AssertTrue(q_Output,
    'Beam within limits, FFO should be true');
    
    
//Req eV moved out of range
stCurBeamParams.neVRange := F_eVRangeCalculator(800, 0);
    
stMachineTargetBeamParams.neVRange := F_eVRangeCalculator(800, 0);

stReqBeamParams.neVRange := 2#0000_1111_0011_1111;

fbPEW.i_xReset := FALSE; //release local FF reset req    
fbPEW(i_stCurrentBeamParams := stCurBeamParams,
    i_stMachineTargetBeamParams := stMachineTargetBeamParams,
    i_stRequestedBeamParams := stReqBeamParams,
    io_fbFFHWO := fbFFO);
    
fbFFO.EvaluateOutput(q_xFastFaultOut=>q_Output);

AssertFalse(q_Output,
    'Limits moved beyond current and target beam, should produce a fault.');

//Beam and target eV moved back within permitted ranges, reset clears fault
stCurBeamParams.neVRange := F_eVRangeCalculator( 300, 0);
    
stMachineTargetBeamParams.neVRange := F_eVRangeCalculator(300, 0);

stReqBeamParams.neVRange := 2#0000_1111_0011_1111;

fbFFO(i_xReset:=TRUE); //New reset request

fbPEW.i_xReset := TRUE; //New reset request

fbPEW(i_stCurrentBeamParams := stCurBeamParams, //Beam params are now within spec
    i_stMachineTargetBeamParams := stMachineTargetBeamParams,
    i_stRequestedBeamParams := stReqBeamParams,
    io_fbFFHWO := fbFFO);
    
fbFFO.EvaluateOutput(q_xFastFaultOut=>q_Output);

AssertTrue(q_Output,
    'Beam within limits after reset, FFO should be true');
    
//At this point, the fast fault would be cleared

//Current beam eV moved out of range
stCurBeamParams.neVRange := F_eVRangeCalculator(800, 0); //Moved out of range
    
stMachineTargetBeamParams.neVRange := F_eVRangeCalculator(300, 0); //Still within range

stReqBeamParams.neVRange := 2#0000_1111_0011_1111;

fbPEW(i_stCurrentBeamParams := stCurBeamParams,
    i_stMachineTargetBeamParams := stMachineTargetBeamParams,
    i_stRequestedBeamParams := stReqBeamParams,
    io_fbFFHWO := fbFFO);
    
fbFFO.EvaluateOutput(q_xFastFaultOut=>q_Output);

AssertFalse(q_Output,
    'Current beam moved beyond set limits, should produce a fault');

//Target beam eV moved out of range
fbFFO(i_xReset:=FALSE); //Reset released
fbFFO(i_xReset:=TRUE); //New reset request comes in at the top of a cycle, but will be overridden

stCurBeamParams.neVRange := F_eVRangeCalculator(300, 0); //Now within range
    
stMachineTargetBeamParams.neVRange := F_eVRangeCalculator(800, 0); //Moved out of range

stReqBeamParams.neVRange := 2#0000_1111_0011_1111;

fbPEW.i_xReset := TRUE; //Attempt to reset local FF will fail
fbPEW(i_stCurrentBeamParams := stCurBeamParams,
    i_stMachineTargetBeamParams := stMachineTargetBeamParams,
    i_stRequestedBeamParams := stReqBeamParams,
    io_fbFFHWO := fbFFO);
    
fbFFO.EvaluateOutput(q_xFastFaultOut=>q_Output);

AssertFalse(q_Output,
    'Target beam moved beyond set limits, should produce a fault');
    
TEST_FINISHED();
END_METHOD

END_FUNCTION_BLOCK

// TestComponents/FB_SafeBPCompare_Test
{attribute 'call_after_init'}
FUNCTION_BLOCK FB_SafeBPCompare_Test EXTENDS TcUnit.FB_TestSuite
VAR_INPUT
END_VAR
VAR_OUTPUT
END_VAR
VAR

END_VAR

BeamOffIsSafe();
BPComparisonCheck();

//Verify beam off is considered safe.
METHOD BeamOffIsSafe
VAR_INPUT
END_VAR
VAR
    stBeamOn_MoreConservative    :    ST_BeamParams;
    stBeamOff_LessConservative    :    ST_BeamParams;
END_VAR
stBeamOn_MoreConservative  := F_SetBeamParams(
    0, //0% transmission is more conservative than 50
    16#FFFF_FFFF,
    120, //rate
    PMPS_GVL.DUMMY_AUX_ATT_ARRAY);

stBeamOff_LessConservative:= F_SetBeamParams(
    0.5, //50% transmission, less conservative, without 0-rate this beam parameter set would be less safe than above
    16#FFFF_FFFF,
    0, //rate, hence, more conservative
    PMPS_GVL.DUMMY_AUX_ATT_ARRAY); //0 beam rate means this bps is actually safer than BeamOn

TEST('BeamOffIsSafe');
    
AssertTrue(
    F_SafeBPCompare0Rate(stBeamOff_LessConservative, stBeamOn_MoreConservative),
    'SafeBPCompare does not think beam rate = 0 is safer than anything else.'); 
TEST_FINISHED();
END_METHOD

//Verify BP comparison remains logical.
METHOD BPComparisonCheck
VAR_INPUT
END_VAR
VAR
    stSafer    :    ST_BeamParams;
    stNotSoSafe    :    ST_BeamParams;
    idx : UINT;
    
    xResult : BOOL;
    xFailedTest : BOOL; // To exit loops early
END_VAR

TEST('BPComparisonTran');
//Attenuation
stSafer := F_SetBeamParams(
    0.51, //
    16#FFFFFFFF,
    1,
    PMPS_GVL.DUMMY_AUX_ATT_ARRAY);

stNotSoSafe := F_SetBeamParams(
    0.61, //
    16#FFFFFFFF,
    1,
    PMPS_GVL.DUMMY_AUX_ATT_ARRAY); 
    
AssertTrue(
    F_SafeBPCompare(stSafer, stNotSoSafe),
    'Attenuation eval is broken (True)'); 

AssertFalse(
    F_SafeBPCompare(stNotSoSafe, stSafer),
    'Attenuation eval is broken (False)');
    
// Check at margin threshold
stSafer.nTran := stNotSoSafe.nTran*(PMPS_GVL.TRANS_SCALING_FACTOR + PMPS_PARAM.TRANS_MARGIN)/PMPS_GVL.TRANS_SCALING_FACTOR;
AssertTrue(
    F_SafeBPCompare(stSafer, stNotSoSafe),
    'Attenuation eval is broken: should be safe up to margin.');

stSafer.nTran := 1 + stNotSoSafe.nTran*(PMPS_GVL.TRANS_SCALING_FACTOR + PMPS_PARAM.TRANS_MARGIN)/PMPS_GVL.TRANS_SCALING_FACTOR;

AssertFalse(
    F_SafeBPCompare(stSafer, stNotSoSafe),
    'Attenuation eval is broken (False): should not be safe at all past margin');

TEST_FINISHED();


    
//Attenuator array    
TEST('BPComparisonTranArray');

stSafer := F_SetBeamParams(
    0, //
    16#FFFFFFFF,
    1,
    PMPS_GVL.DUMMY_AUX_ATT_ARRAY); 

stNotSoSafe := F_SetBeamParams(
    0, //
    16#FFFFFFFF,
    1,
    PMPS_GVL.DUMMY_AUX_ATT_ARRAY); 

FOR idx:=1 TO PMPS_GVL.AUX_ATTENUATORS DO
    stSafer.astAttenuators[idx].nTran := 0.00500;
    stNotSoSafe.astAttenuators[idx].nTran := 0.00600;
    
    xResult := F_SafeBPCompare(stSafer, stNotSoSafe);
    
    AssertTrue(
    xResult,
    'Attenuation array eval is broken (True)');
 
    xFailedTest S= NOT xResult;
    
    xResult := F_SafeBPCompare(stNotSoSafe, stSafer);
    AssertFalse(
    xResult,
    'Attenuation array eval is broken (False)');
    
    xFailedTest S= xResult;
    
    // Check at margin threshold
        stSafer.astAttenuators[idx].nTran := stNotSoSafe.astAttenuators[idx].nTran*(PMPS_GVL.TRANS_SCALING_FACTOR + PMPS_PARAM.TRANS_MARGIN)/PMPS_GVL.TRANS_SCALING_FACTOR;
        
        xResult := F_SafeBPCompare(stSafer, stNotSoSafe);
    
        AssertTrue(
            xResult,
            'Attenuation eval is broken: should be safe up to margin.');
        xFailedTest S= NOT xResult;
            
        stSafer.astAttenuators[idx].nTran := 1 + stNotSoSafe.astAttenuators[idx].nTran*(PMPS_GVL.TRANS_SCALING_FACTOR + PMPS_PARAM.TRANS_MARGIN)/PMPS_GVL.TRANS_SCALING_FACTOR;
        
        xResult := F_SafeBPCompare(stSafer, stNotSoSafe);
        AssertFalse(
            xResult,
            'Attenuation eval is broken (False): should not be safe at all past margin');
        xFailedTest S= xResult;
    //////////////////////
    IF xFailedTest THEN
        stSafer.astAttenuators[idx].nTran := 0;
        stNotSoSafe.astAttenuators[idx].nTran := 0;
        xFailedTest := FALSE;
        EXIT; // Exit this loop on the first failure.
	END_IF
    
    stSafer.astAttenuators[idx].nTran := 0;
    stNotSoSafe.astAttenuators[idx].nTran := 0;
    
END_FOR

TEST_FINISHED();

stSafer.astAttenuators[idx].nTran := 0;
stNotSoSafe.astAttenuators[idx].nTran := 0;

//Aperture array
TEST('BPComparisonApertureArray');

FOR idx:=1 TO PMPS_GVL.MAX_APERTURES DO
    // Height
    stSafer.astApertures[idx].Height := 30; // narrower is safer
    stNotSoSafe.astApertures[idx].Height := 50;
    
    AssertTrue(
    F_SafeBPCompare(stSafer, stNotSoSafe),
    'Aperture array eval is broken on height (True)'); 

    AssertFalse(
    F_SafeBPCompare(stNotSoSafe, stSafer),
    'Aperture array eval is broken on height (False)');
    
    IF NOT F_SafeBPCompare(stSafer, stNotSoSafe) or F_SafeBPCompare(stNotSoSafe, stSafer) THEN
        EXIT; // Exit this loop on the first failure.
	END_IF
    
    stSafer.astApertures[idx].Height := 0;
    stNotSoSafe.astApertures[idx].Height := 0;
    
    // Width
    stSafer.astApertures[idx].Width := 30; // narrower is safer
    stNotSoSafe.astApertures[idx].Width := 50;
    
    AssertTrue(
    F_SafeBPCompare(stSafer, stNotSoSafe),
    'Aperture array eval is broken on width (True)'); 

    AssertFalse(
    F_SafeBPCompare(stNotSoSafe, stSafer),
    'Aperture array eval is broken on width (False)');
    
    IF NOT F_SafeBPCompare(stSafer, stNotSoSafe) or F_SafeBPCompare(stNotSoSafe, stSafer) THEN
        EXIT; // Exit this loop on the first failure.
	END_IF
    
    stSafer.astApertures[idx].Width := 0;
    stNotSoSafe.astApertures[idx].Width := 0;
    
    
END_FOR

TEST_FINISHED();
    
//Rate
TEST('BPComparisonRate');
stSafer := F_SetBeamParams(
    0,
    16#FFFF_FFFF,
    1,
    PMPS_GVL.DUMMY_AUX_ATT_ARRAY); //

stNotSoSafe := F_SetBeamParams(
    0,
    16#FFFF_FFFF,
    10,
    PMPS_GVL.DUMMY_AUX_ATT_ARRAY); //
    
AssertTrue(
    F_SafeBPCompare(stSafer, stNotSoSafe),
    'Rate eval is broken (True)'); 

AssertFalse(
    F_SafeBPCompare(stNotSoSafe, stSafer),
    'Rate eval is broken (False)');
TEST_FINISHED();
    
//Pulse energy
(*
TEST('BPComparisonPulseEnergy');
stSafer := F_SetBeamParams(
    0, 
    1, //
    16#FFFF,
    1,
    PMPS_GVL.DUMMY_AUX_ATT_ARRAY);

stNotSoSafe := F_SetBeamParams(
    0, 
    10, //
    16#FFFF,
    1,
    PMPS_GVL.DUMMY_AUX_ATT_ARRAY); 
    *)
AssertTrue(
    F_SafeBPCompare(stSafer, stNotSoSafe),
    'Pulse energy eval is broken (True)'); 

AssertFalse(
    F_SafeBPCompare(stNotSoSafe, stSafer),
    'Pulse energy eval is broken (False)');    
TEST_FINISHED();
    
//Photon energy
//More extensive tests elsewhere
TEST('BPComparisonPhotonEnergy');
stSafer := F_SetBeamParams(
    0, 
    2#0000_0000_0000_0000_0000_0000_0000_0010,
    1,
    PMPS_GVL.DUMMY_AUX_ATT_ARRAY);

stNotSoSafe := F_SetBeamParams(
    0, 
    2#0000_0000_0000_0000_0000_0000_0000_0110,
    1,
    PMPS_GVL.DUMMY_AUX_ATT_ARRAY);
    
AssertTrue(
    F_SafeBPCompare(stSafer, stNotSoSafe),
    'Photon energy eval is broken (True)'); 

AssertFalse(
    F_SafeBPCompare(stNotSoSafe, stSafer),
    'Photon energy eval is broken (False)');    
TEST_FINISHED();
END_METHOD

END_FUNCTION_BLOCK

// TestComponents/FB_SubsysToArb_Test
{attribute 'call_after_init'}
FUNCTION_BLOCK FB_SubsysToArb_Test EXTENDS TcUnit.FB_TestSuite
VAR_INPUT
END_VAR
VAR_OUTPUT
END_VAR
VAR
END_VAR

BasicFunction();
VetoFunction();

METHOD BasicFunction
VAR_INPUT
END_VAR
VAR   
    nId    :    DWORD := 1;
    stReq    :    ST_BeamParams := (nTran:=12);
END_VAR
VAR_INST
    fbArbiter    :    FB_Arbiter(1);
    
    fbSubSysToArb : FB_SubSysToArbiter_IO; // Subsystem interface with beamline arbiter PLC
    pBPC : POINTER TO ST_BeamParams_IO;
    
    ioCurrentBP : ST_BeamParams_IO; 
    
    FFO : FB_HardwareFFOutput; // Dummy FFO not important for these tests
    
    nCohortScratch : UDINT;
    
END_VAR
VAR CONSTANT
    SysID : DWORD := 42;
END_VAR
// This simulates a synchronous cycle between the subsystem and arbiter PLC cycles. Ie. phase is locked, and cycle time is the same. This is not always the case, so these tests should be 
// trusted with a grain of salt.

TEST('Add to arbiter');

IF NOT fbArbiter.CheckRequestInPool(nID) THEN
    AssertTrue(fbArbiter.AddRequest(nId, stReq,'Device'), 'Arbiter returned false from AddRequest'); // some device asking its local arbiter for some beam parameters
END_IF  
   
TEST_FINISHED();   

///////////////////////////////////////
//Sub system cycle
fbSubSysToArb(Arbiter := fbArbiter, fbFFHWO := FFO);
//END of sub system cycle
///////////////////////////////////////


TEST('Initial Elevation');
AssertTrue(fbSubSysToArb.nRequestCohort = fbSubSysToArb.q_stRequestedBP.nCohortInt, 'ReqCohort and qBP Cohort do not match');
AssertFalse(fbArbiter.nActiveCohort <> 0, 'Arbiter indicates it is included in arbitration prematurely');
AssertTrue(fbSubSysToArb.nRequestCohort <> 0, 'Cohort index should move to 1 with first request');
TEST_FINISHED_NAMED('Initial Elevation');

nCohortScratch := fbSubSysToArb.nRequestCohort;
    
//Ethercat transfer simulation
// Transfer of requested BP to arbiter PLC
// pBPR := ADR(fbArbToSubSys.i_RequestedBP);
// pBPR^ := fbSubSysToArb.q_stRequestedBP;

ioCurrentBP := fbSubSysToArb.q_stRequestedBP;
// NOTE: Setting the returning cohort number to something less than the request cohort number
// will prevent the sub system arbiter FB from considering itself active in arbitration.
// The next set of tests verify this.
ioCurrentBP.nCohortInt := 0;

// Transfer of current BP to sub system PLC
pBPC := ADR(fbSubSysToArb.i_stCurrentBP);
pBPC^ := ioCurrentBP;

///////////////////////////////////////
//Sub system cycle
fbSubSysToArb(Arbiter := fbArbiter, fbFFHWO := FFO);
//END of sub system cycle
///////////////////////////////////////

TEST('Not yet active in arbitration');
AssertTrue(fbSubSysToArb.nActiveCohort = 0, 'Active cohort should still be zero, per ioCurrentBP.nCohortInt setting above.');
AssertFalse(fbArbiter.nActiveCohort <> 0, 'Arbiter indicates it is included in arbitration prematurely, checkrequest might be broken');
AssertTrue(fbSubSysToArb.nRequestCohort = nCohortScratch, 'Cohort index should not have changed because there have been no additional requests added to the arbiter');
TEST_FINISHED_NAMED('Not yet active in arbitration');

//Ethercat transfer simulation
// Transfer of requested BP to arbiter PLC
// pBPR := ADR(fbArbToSubSys.i_RequestedBP);
// pBPR^ := fbSubSysToArb.q_stRequestedBP;

ioCurrentBP := fbSubSysToArb.q_stRequestedBP;
// NOTE: Now we simulate the FB_ArbiterToSubSys_IO updating the cohort number to the same value as the request cohort, indicating that cohort has been included
ioCurrentBP.nCohortInt := 2;

// Transfer of current BP to sub system PLC
pBPC := ADR(fbSubSysToArb.i_stCurrentBP);
pBPC^ := ioCurrentBP;

///////////////////////////////////////
//Sub system cycle
fbSubSysToArb(Arbiter := fbArbiter, fbFFHWO := FFO);
//END of sub system cycle
///////////////////////////////////////

TEST('Active in arbitration');
AssertTrue(fbSubSysToArb.nActiveCohort = fbSubSysToArb.nRequestCohort, 'Active cohort and request cohort do not match');
AssertTrue(fbArbiter.nActiveCohort = 1, 'Arbiter does not indicate it is included in higher arbitration');
TEST_FINISHED_NAMED('Active in arbitration');
END_METHOD

METHOD VetoFunction
VAR_INPUT
END_VAR
VAR   
    nId    :    DWORD := 1;
    stReq    :    ST_BeamParams := (nTran:=12);
END_VAR
VAR_INST
    fbArbiter    :    FB_Arbiter(1);
    
    fbSubSysToArb : FB_SubSysToArbiter_IO; // Subsystem interface with beamline arbiter PLC
    fbArbToSubSys : FB_ArbiterToSubSys_IO;
    
    pBPC : POINTER TO ST_BeamParams_IO;
    pBPR : POINTER TO ST_BeamParams_IO;
    
    ioCurrentBP : ST_BeamParams_IO; 
    
    FFO : FB_HardwareFFOutput; // Dummy FFO not important for these tests
    
END_VAR
VAR CONSTANT
    SysID : DWORD := 42;
END_VAR
// This simulates a synchronous cycle between the subsystem and arbiter PLC cycles. Ie. phase is locked, and cycle time is the same. This is not always the case, so these tests should be 
// trusted with a grain of salt.

fbArbiter.AddRequest(nId, stReq,'Device'); // some device asking its local arbiter for some beam parameters


///////////////////////////////////////
//Sub system cycle
fbSubSysToArb(Arbiter := fbArbiter, fbFFHWO := FFO);
//END of sub system cycle
///////////////////////////////////////

TEST('Request propagated');
    AssertTrue(fbSubSysToArb.q_stRequestedBP.nTran = stReq.nTran, 'Request not propagated');
TEST_FINISHED();

// Veto activated
///////////////////////////////////////
//Sub system cycle
fbSubSysToArb(Arbiter := fbArbiter, fbFFHWO := FFO, i_bVeto:=TRUE);
//END of sub system cycle
///////////////////////////////////////

// Veto activated
///////////////////////////////////////
//Sub system cycle
fbSubSysToArb(Arbiter := fbArbiter, fbFFHWO := FFO, i_bVeto:=TRUE);
//END of sub system cycle
///////////////////////////////////////

TEST('Request sustained');
    AssertTrue(fbSubSysToArb.q_stRequestedBP.nTran = PMPS_GVL.cstFullBeam.nTran, 'Request still being propagated');
    AssertTrue(fbArbiter.CheckRequest(nId), 'Request still not valid');
TEST_FINISHED();

// Veto activated
///////////////////////////////////////
//Sub system cycle
fbSubSysToArb(Arbiter := fbArbiter, fbFFHWO := FFO, i_bVeto:=FALSE);
//END of sub system cycle
///////////////////////////////////////

// Veto activated
///////////////////////////////////////
//Sub system cycle
fbSubSysToArb(Arbiter := fbArbiter, fbFFHWO := FFO, i_bVeto:=FALSE);
fbSubSysToArb(Arbiter := fbArbiter, fbFFHWO := FFO, i_bVeto:=FALSE);
fbSubSysToArb(Arbiter := fbArbiter, fbFFHWO := FFO, i_bVeto:=FALSE);
//END of sub system cycle
///////////////////////////////////////

TEST('Request restored');
    AssertTrue(fbSubSysToArb.q_stRequestedBP.nTran = stReq.nTran, 'Request still being sustained');
TEST_FINISHED();
END_METHOD

END_FUNCTION_BLOCK

// TestComponents/FB_VetoArbiter_Test
{attribute 'call_after_init'}
FUNCTION_BLOCK FB_VetoArbiter_Test EXTENDS TcUnit.FB_TestSuite
VAR_INPUT
END_VAR
VAR_OUTPUT
END_VAR
VAR
END_VAR
VAR CONSTANT
    ArbID : DWORD := 1;
	HigherArbID : DWORD := 2;
END_VAR

VetoArbiter();

METHOD VetoArbiter

VAR_INPUT
END_VAR
VAR   
    nId    :    DWORD := 1;
	nId2 : DWORD := 10;
    stReq    :    ST_BeamParams := (nTran:=0.12);
	stReq2	:	ST_BeamParams := (nTran:=0.10);
END_VAR
VAR_INST
    fbArbiter    :    FB_Arbiter(1);
    
    fbHigherArb : FB_Arbiter(2);
	
	ArbBP : ST_BeamParams;
	
	VetoArb : FB_VetoArbiter;
	
	FFO : FB_HardwareFFOutput;
	
	fbHA : FB_DummyHA;
    
END_VAR

TEST('VetoNotIn');
fbArbiter.AddRequest(nReqID:=nId, stReqBP:=stReq, sDevName :='Device');

//////////////////// Cycle    
fbHigherArb.ElevateRequest(fbHA);

VetoArb.bVeto := FALSE;
VetoArb(HigherAuthority:=fbHigherArb,
	LowerAuthority:=fbArbiter,
	FFO:=FFO);
    
//////////////////// Cycle    
fbHigherArb.ElevateRequest(fbHA);

VetoArb.bVeto := FALSE;
VetoArb(HigherAuthority:=fbHigherArb,
	LowerAuthority:=fbArbiter,
	FFO:=FFO);

AssertTrue(fbHigherArb.q_stBeamParams.nTran = stReq.nTran, 'We should see the transmission number here, veto device is not in');

TEST_FINISHED();

TEST('VetoIn');
// Veto device is in
// This should effectively remove the fbArbiter request from the higher arbiter pool

//////////////////// Cycle    
fbHigherArb.ElevateRequest(fbHA);

VetoArb.bVeto := TRUE;
VetoArb(HigherAuthority:=fbHigherArb, // Veto removed
	LowerAuthority:=fbArbiter,
	FFO:=FFO);

//////////////////// Cycle    
fbHigherArb.ElevateRequest(fbHA);

VetoArb.bVeto := TRUE;
VetoArb(HigherAuthority:=fbHigherArb, // Veto removed
	LowerAuthority:=fbArbiter,
	FFO:=FFO);
    
AssertTrue(fbHigherArb.q_stBeamParams.nTran = PMPS_GVL.cstFullBeam.nTran, 'Veto device is in, trans should be restored to 100');
AssertTrue(fbArbiter.CheckRequest(nId), 'Request should still be considered valid (1)');
AssertFalse(fbHigherArb.CheckRequest(ArbID), 'Lower arb request should be gone from the higher pool');

TEST_FINISHED();

TEST('AnotherRequest');
// Another request is added, should be approved immediately, and with no effect on the final set
fbArbiter.RequestBP(nReqID := nId2, stReqBP:=stReq2);

//////////////////// Cycle    
fbHigherArb.ElevateRequest(fbHA);

VetoArb.bVeto := TRUE;
VetoArb(HigherAuthority:=fbHigherArb, // Veto removed
	LowerAuthority:=fbArbiter,
	FFO:=FFO);
    
//////////////////// Cycle    
fbHigherArb.ElevateRequest(fbHA);

VetoArb.bVeto := TRUE;
VetoArb(HigherAuthority:=fbHigherArb, // Veto removed
	LowerAuthority:=fbArbiter,
	FFO:=FFO);

AssertTrue(ArbBP.nTran = PMPS_GVL.cstFullBeam.nTran, 'Veto device remained in, trans should still be 100');
AssertTrue(fbArbiter.CheckRequest(nId), 'Request should still be considered valid (2)');
AssertTrue(fbArbiter.CheckRequest(nId2), '2nd Request should be considered valid');

TEST_FINISHED();

TEST('RemoveVeto');
// Removal of veto device, should produce a fault
//////////////////// Cycle    
fbHigherArb.ElevateRequest(fbHA);

VetoArb.bVeto := FALSE;
VetoArb(HigherAuthority:=fbHigherArb, // Veto removed
	LowerAuthority:=fbArbiter,
	FFO:=FFO);

AssertFalse(VetoArb.ffKeepItSecretKeepItSafe.i_xOK, 'Should produce a fast fault at this point because the request is not yet back in the pool');

//////////////////// Cycle  
fbHigherArb.ElevateRequest(fbHA);

VetoArb.bVeto := FALSE;
VetoArb(HigherAuthority:=fbHigherArb, // Veto removed
	LowerAuthority:=fbArbiter,
	FFO:=FFO);

//////////////////// Cycle    
fbHigherArb.ElevateRequest(fbHA);

VetoArb.bVeto := FALSE;
VetoArb(HigherAuthority:=fbHigherArb, // Veto removed
	LowerAuthority:=fbArbiter,
	FFO:=FFO);

//////////////////// Cycle    
fbHigherArb.ElevateRequest(fbHA);

VetoArb.bVeto := FALSE;
VetoArb(HigherAuthority:=fbHigherArb, // Veto removed
	LowerAuthority:=fbArbiter,
	FFO:=FFO);    
    
AssertTrue(VetoArb.ffKeepItSecretKeepItSafe.i_xOK, 'Fault should be gone.');

TEST_FINISHED();
END_METHOD

END_FUNCTION_BLOCK

// MAIN
PROGRAM MAIN
VAR
    fbSetPERanges : PE_Ranges;    

    fbDiffBPTest    :    FB_DiffBP_Test;
    fbBPTMTest    :    FB_BPTM_Test;
    fbSafeBPCompareTest    :    FB_SafeBPCompare_Test;
    ////fbevWithinSpecTest    :    FB_evWithinSpec_Test;
    ////fbPEWTest    :    FB_PhotonEnergyWatcher_Test;
    fbFFTest    :    FB_FastFault_Test;
    fbArbiterTest    :    FB_Arbiter_Test;
	fbVetoArbiterTest : FB_VetoArbiter_Test;
    fbevRangeCalcTest : FB_evRangeCalculator_Test;
    fbSubSysToArbTest : FB_SubsysToArb_Test;
    fbArbToSubSysTest : FB_ArbToSubsys_Test;
END_VAR

TcUnit.RUN();

END_PROGRAM
